{attribute 'GeneratedUsingTerminal: IODEVICETYPE_ETHERCATPROT'}
{attribute addProperty BoxType "IODEVICETYPE_ETHERCATPROT"}
{attribute addProperty Id "ObjectIdAT %I*OTCID4StateAT %I*UINT2SlaveCountAT %I*UINT2"}
{attribute addProperty CRC "714593999"}
{attribute addProperty Size "8"}
TYPE InfoData_2A97D6CF :
STRUCT
	{attribute addProperty Name "ObjectId"}
	ObjectId AT %I* : OTCID;
	{attribute addProperty Name "State"}
	State AT %I* : UINT;
	{attribute addProperty Name "SlaveCount"}
	SlaveCount AT %I* : UINT;
END_STRUCT
END_TYPE

(* stored: Version 1.2.0.0, ProductVersion 3.1.4024.9
   DUT InfoData_2A97D6CF: Id {561b462a-9f2c-4541-85fc-1094056054d3} *)
